{attribute 'GeneratedUsingTerminal: EL7342-0000-0023'}
{attribute addProperty BoxType "EL7342-0000-0023"}
{attribute addProperty Id "EtcSlaveTerminalBaseENC_Status_compact_Channel_1AT %I*ENC_Status_compact_Channel_DC559AB014ENC_Status_compact_Channel_2AT %I*ENC_Status_compact_Channel_DC559AB014DCM_Status_Channel_1AT %I*DCM_Status_Channel_36ED096F11DCM_Status_Channel_2AT %I*DCM_Status_Channel_36ED096F11ENC_Control_compact_Channel_1AT %Q*ENC_Control_compact_Channel_2E82BC435ENC_Control_compact_Channel_2AT %Q*ENC_Control_compact_Channel_2E82BC435DCM_Control_Channel_1AT %Q*DCM_Control_Channel_94BFDFDF4DCM_Velocity_Channel_1AT %Q*DCM_Velocity_Channel_A47A3F412DCM_Control_Channel_2AT %Q*DCM_Control_Channel_94BFDFDF4DCM_Velocity_Channel_2AT %Q*DCM_Velocity_Channel_A47A3F412WcStateAT %I*WcState_9091E0EB2InfoDataAT %I*InfoData_939F71B614"}
{attribute addProperty CRC "2827126288"}
{attribute addProperty Size "88"}
TYPE EL7342_A8828610 EXTENDS EtcSlaveTerminalBase :
STRUCT
	{attribute addProperty Name "ENC_Status_compact_Channel_1"}
	ENC_Status_compact_Channel_1 : ENC_Status_compact_Channel_DC559AB0;
	{attribute addProperty Name "ENC_Status_compact_Channel_2"}
	ENC_Status_compact_Channel_2 : ENC_Status_compact_Channel_DC559AB0;
	{attribute addProperty Name "DCM_Status_Channel_1"}
	DCM_Status_Channel_1 : DCM_Status_Channel_36ED096F;
	{attribute addProperty Name "DCM_Status_Channel_2"}
	DCM_Status_Channel_2 : DCM_Status_Channel_36ED096F;
	{attribute addProperty Name "ENC_Control_compact_Channel_1"}
	ENC_Control_compact_Channel_1 : ENC_Control_compact_Channel_2E82BC43;
	{attribute addProperty Name "ENC_Control_compact_Channel_2"}
	ENC_Control_compact_Channel_2 : ENC_Control_compact_Channel_2E82BC43;
	{attribute addProperty Name "DCM_Control_Channel_1"}
	DCM_Control_Channel_1 : DCM_Control_Channel_94BFDFDF;
	{attribute addProperty Name "DCM_Velocity_Channel_1"}
	DCM_Velocity_Channel_1 : DCM_Velocity_Channel_A47A3F41;
	{attribute addProperty Name "DCM_Control_Channel_2"}
	DCM_Control_Channel_2 : DCM_Control_Channel_94BFDFDF;
	{attribute addProperty Name "DCM_Velocity_Channel_2"}
	DCM_Velocity_Channel_2 : DCM_Velocity_Channel_A47A3F41;
	{attribute addProperty Name "WcState"}
	WcState : WcState_9091E0EB;
	{attribute addProperty Name "InfoData"}
	InfoData : InfoData_939F71B6;
END_STRUCT
END_TYPE

(* stored: Version 1.2.0.0, ProductVersion 3.1.4024.9
   DUT EL7342_A8828610: Id {7d8d94db-0551-41fa-bdd5-177c73258726} *)
